FUNCTION_BLOCK Dilate (* openCV dilate filter *)
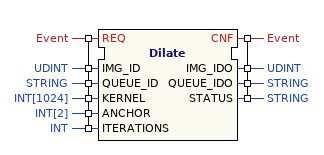
  EVENT_INPUT
    REQ WITH IMG_ID, QUEUE_ID, KERNEL, ANCHOR, ITERATIONS;
  END_EVENT
  EVENT_OUTPUT
    CNF WITH IMG_IDO, QUEUE_IDO, STATUS;
  END_EVENT
  VAR_INPUT
    IMG_ID : UDINT;
    QUEUE_ID : STRING;
    KERNEL : ARRAY [0..1023] OF INT;
    ANCHOR : ARRAY [0..1] OF INT;
    ITERATIONS : INT;
  END_VAR
  VAR_OUTPUT
    IMG_IDO : UDINT;
    QUEUE_IDO : STRING;
    STATUS : STRING;
  END_VAR
END_FUNCTION_BLOCK
